// TIA Portal V17 export
// export: Created 2026-04-13T11:12:44.3267403Z, ExportSetting WithDefaults, DisplayName Totally Integrated Automation Portal, DisplayVersion V17 Update 4, DisplayName TIA Portal Openness, DisplayVersion V17 Update 4, DisplayName TIA Portal Version Control Interface, DisplayVersion V17, DisplayName SINAMICS Startdrive Advanced, DisplayVersion V17, DisplayName SINAMICS Startdrive G130, G150, S120, S150, SINAMICS MV, S210, DisplayVersion V17, DisplayName SINAMICS Startdrive G110M, G120, G120C, G120D, G120P, G115D, DisplayVersion V17, DisplayName STEP 7 Professional, DisplayVersion V17 Update 4, DisplayName STEP 7 Safety, DisplayVersion V17, DisplayName WinCC Professional, DisplayVersion V17 Update 4
DATA_BLOCK "A4-脉冲控制_DB"   // DB4
VERSION : 0.1
// stored: AutoNumber true, DBAccessibleFromOPCUA true, DBAccessibleFromWebserver true, InstanceOfName A4-脉冲控制, InstanceOfType FB
"A4-脉冲控制"
   // VAR
   //    主塔气锤 { S7_SetPoint := 'True'} : "A3-脉冲轮询";
   //    二级旋风振打锤 { S7_SetPoint := 'True'} : "A3-脉冲轮询";
   //    一级旋风振打锤 { S7_SetPoint := 'True'} : "A3-脉冲轮询";
   //    一级旋风振荡器 { S7_SetPoint := 'True'} : "A3-脉冲轮询";
   //    布袋气锤 { S7_SetPoint := 'True'} : "A3-脉冲轮询";
   //    布袋反吹 { S7_SetPoint := 'True'} : "A3-脉冲轮询";
   //    设备振打 { S7_SetPoint := 'True'} : "A3-脉冲轮询";
   //    输送出料 { S7_SetPoint := 'True'} : "A3-脉冲轮询";
   //    布袋出料 { S7_SetPoint := 'True'} : "A3-脉冲轮询";
   //    一级旋风出料 { S7_SetPoint := 'True'} : "A3-脉冲轮询";
   //    二级旋风出料 { S7_SetPoint := 'True'} : "A3-脉冲轮询";
   //    布袋出料1 { S7_SetPoint := 'True'} : "A9-循环下料控制";
   //    一级旋风出料1 { S7_SetPoint := 'True'} : "A9-循环下料控制";
   //    二级旋风出料1 { S7_SetPoint := 'True'} : "A9-循环下料控制";
   //    LT1 : Real;
   // END_VAR
BEGIN
END_DATA_BLOCK
